// TIA Portal V20 export
TYPE "LConSMC_typeAxisCyclicData"
// stored: Access Published
   STRUCT
      actualSpeed : LReal;
      velocity : LReal;
      actualTorque : LReal;
      actualPosition : LReal;
   END_STRUCT;
END_TYPE
